(*
SPDX-FileCopyrightText: © 2026 Oleksandr Tiutyk <trofimich@gmail.com>
SPDX-License-Identifier: MIT
License: https://opensource.org/license/mit
*)

TYPE AUTOMATION_ERROR_LOG :
STRUCT
	ShortMessage : TOF_Core.ERROR_MESSAGE;
	FullMessage : TOF_Core.ERROR_MESSAGE;
	Source : STRING(255);
	LocalTimestamp : LDATE_AND_TIME;	
	UtcTimestamp : LDATE_AND_TIME;	
END_STRUCT
END_TYPE

(* stored: Version 1.1.0.1
   DUT AUTOMATION_ERROR_LOG: Id {43dcf754-537c-4e04-b7ec-3c711cbf3a59} *)
